PROGRAM SEQ_CR_PLACE
VAR_INPUT
	CR_Place_Rack	: UINT;
	CR_found		: BOOL;
END_VAR
VAR
	CR_place_num 	: UINT;
END_VAR

// Get next CR POS
IF NOT CR_found THEN
//	FOR CR_place_num := GVL.CR_NextPlaceNum TO 6 BY 1 DO
	FOR CR_place_num := 2 TO 21 BY 1 DO
		IF GVL.CR_NextPlaceNum > 21 OR GVL.CR_NextPlaceNum < 2 THEN
			GVL.CR_NextPlaceNum := CR_place_num := 2;
		END_IF
		IF GVL.CR_NextPlaceNum = 14 OR GVL.CR_NextPlaceNum = 8 OR GVL.CR_NextPlaceNum = 15 THEN
			GVL.CR_NextPlaceNum := GVL.CR_NextPlaceNum+1;
		ELSIF NOT COOL_RACK.CR[CR_place_num] THEN
			CR_Place_Rack		:= CR_place_num;
			GVL.CR_NextPlaceNum := CR_place_num +1 ;
			CR_found 			:= TRUE;
			RETURN;
		END_IF
	END_FOR
END_IF

END_PROGRAM

(* stored: Version 1.1.0.1, ProductVersion 3.1.4024.12
   POU SEQ_CR_PLACE: Id {ca0f8682-d030-419b-8cfe-0f9c6e0bf6f3}, SpecialFunc None *)
